Fanuc TP program (LS listing): test_home.ls

/PROG  TEST_HOME
/ATTR
OWNER		= MNEDITOR;
COMMENT		= "";
PROG_SIZE	= 525;
CREATE		= DATE 26-05-08  TIME 15:17:14;
MODIFIED	= DATE 26-05-08  TIME 15:17:14;
FILE_NAME	= TEST_HOM;
VERSION		= 0;
LINE_COUNT	= 3;
MEMORY_SIZE	= 885;
PROTECT		= READ_WRITE;
TCD:  STACK_SIZE	= 0,
      TASK_PRIORITY	= 50,
      TIME_SLICE	= 0,
      BUSY_LAMP_OFF	= 0,
      ABORT_REQUEST	= 0,
      PAUSE_REQUEST	= 0;
DEFAULT_GROUP	= 1,*,*,*,*;
CONTROL_CODE	= 00000000 00000000;
LOCAL_REGISTERS	= 0,0,0;
/APPL
/APPL
/MN
   1:  UFRAME_NUM=1 ;
   2:  UTOOL_NUM=1 ;
   3:J PR[1:TMP_DATUM] 100% FINE    ;
/POS
P[1:"HOME"]{
   GP1:
	UF : 1, UT : 1,		CONFIG : 'L, 0, 0, 0',
	X =     0.000000  mm,	Y =     0.000000  mm,	Z =     0.000000  mm,
	W =     0.000000 deg,	P =     0.000000 deg,	R =     0.000000 deg
};
/END
